# EPICS autosave request: autosave/request_files/autosave_ITBL_PROC.req
# ITBL
$(Sec)-$(Sub):$(Dis)-$(Dev)$(Idx):ITBL.VAL
